FUNCTION_BLOCK BrokenCalculator IMPLEMENTS ISum

(*This method adds two DINT numbers and returns the result in Sum*)
METHOD Sum : DINT
VAR_INPUT
	Dint1 : DINT;
	Dint2 : DINT;
END_VAR
Sum := Dint1 * Dint2;
END_METHOD

END_FUNCTION_BLOCK

(* stored: Version 1.1.0.1, ProductVersion 3.1.4024.6
   POU BrokenCalculator: Id {6503d53b-0719-4282-bbb7-efb4ef797492}, SpecialFunc None
   Method Sum: Id {3d36953f-2065-4b1a-bf50-4e1589a6f50b} *)
